KUKA KRL program: GUN_OPEN_CHECK.src, gun_open_check.dat

--- GUN_OPEN_CHECK.src ---
&ACCESS RVO1
&REL 2
&COMMENT 03-10-R1 PNW1 GUN OPEN CHECK
&PARAM EDITMASK = *
&PARAM TEMPLATE = C:\KRC\Roboter\Template\vorgabe
DEF GUN_OPEN_CHECK( )
;********************************
; Gestamp Standards
; Line - BMW G65 (cell 03)
; Robot 03-10-R1 (BMW-03-10-R1-PNW1)
; Application - NUT WELDER GUN OPEN INTERLOCK BEFORE THE ROBOT MOVES INTO OR OUT OF THE PEDESTAL
;********************************
; CALLED BY style1app1opt1..3 BEFORE ENTERING THE PEDESTAL AND BY CENTERLINE_WELD AFTER THE GUN
; OPENS. CHECKS IN THIS ORDER, EACH WITH A STATE MESSAGE AND A WAIT (THE ROBOT DOES NOT MOVE):
; 1. SUBMIT RUNNING ($PRO_STATE0): CL_GunStrokePositionLPT IS ONLY UPDATED BY SPS.SUB
; 2. AIR PRESSURE - SIGNAL $IN[3132] dipw1_AirOK ON (ONLY WITH bGunAirCheck TRUE)
; 3. COOLING WATER - dipw1_WaterOk (SET BY SPS.SUB FROM THE SV0500 FLOW, ONLY WITH bGunWaterCheck)
; 4. GUN OPEN - CL_GunStrokePositionLPT IN nGunOpenMin..nGunOpenMax, nGunOpenWaitMs WITHOUT MESSAGE
; GUN_OPEN_LOST (BELOW) IS THE ROUTINE OF THE GUN MONITORING INTERRUPTS 20-22 OF THE WELD APPS.
; SETTINGS IN GUN_OPEN_CHECK.dat. WRITTEN BY THE PROGRAMMER ON 2026-10-05 (F01)
;CHECK: CLAMP OPEN $IN[466] AND QFP RETURNED $IN[482] ARE NOT CHECKED BEFORE ENTERING (F01)
DECL KrlMsg_T Msg
DECL KrlMsg_T MsgW
DECL KrlMsgPar_T Par[3]
DECL KrlMsgOpt_T Opt
DECL INT nHandle, nWaitMs
DECL BOOL bRes

   ;STOP THE ADVANCE RUN: THE GUN POSITION IS READ WITH THE ROBOT STOPPED, NOT AHEAD OF THE MOTION
   WAIT SEC 0

   ;FOLD MESSAGE SETUP
   Msg.Modul[]="GunOpenCheck"
   MsgW.Modul[]="GunOpenCheck"
   Par[1].Par_Type=#EMPTY
   Par[2].Par_Type=#EMPTY
   Par[3].Par_Type=#EMPTY
   Opt.VL_Stop=TRUE
   Opt.Clear_P_Reset=TRUE
   Opt.Clear_P_SAW=FALSE
   Opt.Log_To_DB=TRUE
   ;ENDFOLD

   ;1. SUBMIT RUNNING - OTHERWISE CL_GunStrokePositionLPT IS FROZEN (NO TIMEOUT, STATE MESSAGE)
   IF $PRO_STATE0<>#P_ACTIVE THEN
      Msg.Nr=1
      Msg.Msg_txt[]="Submit (SPS) not running - gun position not valid - robot waiting"
      Par[1].Par_Type=#EMPTY
      nHandle=Set_KrlMsg(#STATE, Msg, Par[], Opt)
      WAIT FOR $PRO_STATE0==#P_ACTIVE
      bRes=Clear_KrlMsg(nHandle)
      ;LET THE SUBMIT REFRESH THE GUN POSITION
      WAIT SEC 0.5
   ENDIF

   ;2. AIR PRESSURE - WITHOUT AIR THE GUN CANNOT BE HELD OPEN (ONLY WITH bGunAirCheck TRUE)
   IF bGunAirCheck THEN
      ;AIR PRESSURE SWITCH - SIGNAL $IN[3132] dipw1_AirOK ON, ELSE MESSAGE AND WAIT (NO TIMEOUT)
      IF NOT dipw1_AirOK THEN
         Msg.Nr=3
         Msg.Msg_txt[]="Nut welder air pressure not OK (dipw1_AirOK) - robot waiting"
         Par[1].Par_Type=#EMPTY
         nHandle=Set_KrlMsg(#STATE, Msg, Par[], Opt)
         WAIT FOR dipw1_AirOK
         bRes=Clear_KrlMsg(nHandle)
      ENDIF
   ENDIF

   ;3. COOLING WATER - dipw1_WaterOk FROM THE SV0500 FLOW (SPS.SUB); MESSAGE WITH THE FLOW, WAIT
   IF bGunWaterCheck THEN
      IF NOT dipw1_WaterOk THEN
         MsgW.Nr=6
         MsgW.Msg_txt[]="Nut welder cooling water flow too low (%1 x0.1 l/min) - robot waiting"
         Par[1].Par_Type=#VALUE
         Par[1].Par_Int=nWaterFlow
         nHandle=Set_KrlMsg(#STATE, MsgW, Par[], Opt)
         WAIT FOR dipw1_WaterOk
         bRes=Clear_KrlMsg(nHandle)
         Par[1].Par_Type=#EMPTY
      ENDIF
   ENDIF

   ;4. GUN OPEN - UP TO nGunOpenWaitMs WITHOUT MESSAGE
   nWaitMs=0
   WHILE ((CL_GunStrokePositionLPT<nGunOpenMin) OR (CL_GunStrokePositionLPT>nGunOpenMax)) AND (nWaitMs<nGunOpenWaitMs)
      WAIT SEC 0.05
      nWaitMs=nWaitMs+50
   ENDWHILE

   ;GUN STILL NOT OPEN - STATE MESSAGE WITH THE POSITION, WAIT (NO TIMEOUT)
   IF (CL_GunStrokePositionLPT<nGunOpenMin) OR (CL_GunStrokePositionLPT>nGunOpenMax) THEN
      Msg.Nr=2
      Msg.Msg_txt[]="Nut welder gun not open (position %1) - robot waiting"
      Par[1].Par_Type=#VALUE
      Par[1].Par_Int=CL_GunStrokePositionLPT
      nHandle=Set_KrlMsg(#STATE, Msg, Par[], Opt)
      WAIT FOR (CL_GunStrokePositionLPT>=nGunOpenMin) AND (CL_GunStrokePositionLPT<=nGunOpenMax)
      bRes=Clear_KrlMsg(nHandle)
   ENDIF

END

GLOBAL DEF GUN_OPEN_LOST( )
;INTERRUPT ROUTINE OF THE GUN MONITORING (INTERRUPTS 20-22 IN style1app1opt1..3): THE GUN LEFT THE
;OPEN RANGE OR THE SUBMIT STOPPED WHILE THE ROBOT MOVES INTO OR OUT OF THE PEDESTAL. BRAKE F STOPS
;THE ROBOT ON ITS PATH; IT CONTINUES WHEN THE QUIT MESSAGE IS ACKNOWLEDGED AND THE GUN IS OPEN AGAIN
DECL KrlMsg_T Msg
DECL KrlMsgPar_T Par[3]
DECL KrlMsgOpt_T Opt
DECL INT nHandle

   BRAKE F

   ;FOLD MESSAGE SETUP
   Msg.Modul[]="GunOpenCheck"
   Par[1].Par_Type=#EMPTY
   Par[2].Par_Type=#EMPTY
   Par[3].Par_Type=#EMPTY
   Opt.VL_Stop=TRUE
   Opt.Clear_P_Reset=TRUE
   Opt.Clear_P_SAW=FALSE
   Opt.Log_To_DB=TRUE
   ;ENDFOLD

   IF $PRO_STATE0<>#P_ACTIVE THEN
      Msg.Nr=5
      Msg.Msg_txt[]="Submit (SPS) stopped while robot in welder - robot stopped, acknowledge"
   ELSE
      Msg.Nr=4
      Msg.Msg_txt[]="Gun not open while robot in welder (pos. %1) - robot stopped, acknowledge"
      Par[1].Par_Type=#VALUE
      Par[1].Par_Int=CL_GunStrokePositionLPT
   ENDIF
   nHandle=Set_KrlMsg(#QUIT, Msg, Par[], Opt)

   ;CONTINUE ONLY WHEN THE MESSAGE IS ACKNOWLEDGED, THE SUBMIT RUNS AND THE GUN IS OPEN AGAIN
   WHILE Exists_KrlMsg(nHandle) OR ($PRO_STATE0<>#P_ACTIVE) OR (CL_GunStrokePositionLPT<nGunOpenMin) OR (CL_GunStrokePositionLPT>nGunOpenMax)
      WAIT SEC 0.1
   ENDWHILE

END

--- gun_open_check.dat ---
&ACCESS  RV
&COMMENT 03-10-R1 PNW1 GUN OPEN CHECK
&PARAM EDITMASK = *
&PARAM TEMPLATE = C:\KRC\Roboter\Template\vorgabe
&REL 2
DEFDAT  GUN_OPEN_CHECK PUBLIC
;FOLD GUN OPEN SETTINGS
;OPEN (RETRACT) RANGE OF THE NUT WELDER GUN ON 03-10-R1, CL_GunStrokePositionLPT (SPS.SUB):
;NOMINAL RETRACT 139815; WELD RANGE CL_GUN_WELD_MIN..CL_GUN_WELD_MAX (69000..73000, GUN CLOSED)
;WARNING: INTERRUPTS 20/21 IN style1app1opt1..3 REPEAT THIS RANGE AS LITERALS - CHANGE BOTH TOGETHER
;NOTE: REPLACES THE OLDER, WIDER CHECK CL_GunStrokePositionLPT > 120000 AT THE END OF CENTERLINE_WELD
DECL GLOBAL INT nGunOpenMin=137000
DECL GLOBAL INT nGunOpenMax=142000
;TIME FOR THE GUN TO OPEN BEFORE THE "GUN NOT OPEN" MESSAGE [MS]
DECL INT nGunOpenWaitMs=2000
;AIR PRESSURE CHECK - SIGNAL $IN[3132] dipw1_AirOK (TBEN BIT 3.4). TRUE = ACTIVE
;CHECK: DISABLED UNTIL TESTED: WITH THE AIR CLOSED $IN[3132] MUST GO OFF, THEN SET TRUE (F01)
DECL BOOL bGunAirCheck=FALSE
;COOLING WATER FLOW (PARKER 5097335, SPS.SUB) IN 0.1 L/MIN: 150 = 15.0 L/MIN (4.0 GPM)
;WATER OK AT OR ABOVE nWaterFlowMin, NOT OK BELOW nWaterFlowMin - nWaterFlowHyst
;CHECK: NORMAL FLOW 23-26 L/MIN WAS MEASURED ON 03-20-R1; CONFIRM THE MINIMUM ON THIS ROBOT (F09)
DECL GLOBAL INT nWaterFlow=226
DECL GLOBAL INT nWaterFlowMin=150
DECL GLOBAL INT nWaterFlowHyst=10
;COOLING WATER CHECK BEFORE ENTERING / LEAVING THE PEDESTAL. TRUE = ACTIVE
DECL BOOL bGunWaterCheck=TRUE
;ENDFOLD
ENDDAT
